(************************************************************************************************************)
(*							Beckhoff Automation Poland														*)
(*								FB_TypeJK_Sel  v1															*)
(*									27.05.2008																*)
(*	Bloczek przerzutnika JK z uzyciem funckji SEL(select)													*)
(*	Przerzutnik ma wejścia informacyjne (J i K), , wyjście proste (Q) i jego negację (nie Q),				*)
(*	Przerzutnik jest przerzutnikiem synchronicznym, co oznacza, że zmienia stan przy zmianie stanu wejścia 	*)
(*	zegarowego z niskiego na wysoki (0 na 1)-wyzwalanie zboczem narastającym lub przy zmianie stanu			*)
(*	wejścia zegarowego(CLK) z wysokiego na niski (1 na 0)- wyzwalanie zboczem opadającym .					*)
(*	Stan wyjść podczas pracy przerzutnika zależy od stanu wejść, jak i stanu poprzedniego wyjść.			*)
(*__________________________________________________________________________________________________________*)
FUNCTION_BLOCK FB_TypeJK_SEL
VAR_INPUT
	J:			BOOL;
	Clk:		BOOL;
	K:			BOOL;
END_VAR
VAR_OUTPUT
	Q:			BOOL;
END_VAR
VAR
	lastClk:	BOOL;
	lastQ: 		BOOL;
END_VAR

IF (lastClk<Clk) THEN
	Q:=SEL(J=1 AND K=0,Q,FALSE);
	Q:=SEL(J=0 AND K=1,Q,TRUE);
	Q:=SEL(J=1 AND K=1,Q,NOT lastQ);
	Q:=SEL(J=0 AND K=0,Q,lastQ);
END_IF
lastQ:=Q;
lastClk:=Clk;

END_FUNCTION_BLOCK

(* stored: Version 1.1.0.1, ProductVersion 3.1.4020.3
   POU FB_TypeJK_SEL: Id {768cfe6d-3520-4721-a058-ea164f7ac78a}, SpecialFunc None *)
